FUNCTION_BLOCK TcoDrivesBeckhoffContext EXTENDS TcoCore._internals_TcoContext
VAR
	_callMyPlcInstance 		:	BOOL := FALSE;
	_axis					:	TcoDriveSimpleTest(THIS^);
	_enable					:	BOOL;			
	_enablePositive			:	BOOL;				
	_enableNegative			:	BOOL;        	
	_calibrationCam 		:	BOOL;        	
END_VAR

IF THIS^._callMyPlcInstance THEN
	THIS^.Run();
END_IF

{attribute 'TcRpcEnable'}
METHOD Axis
VAR_INPUT
END_VAR
_axis(	inEnable			:=	_enable, 
		inEnablePositive	:=	_enablePositive, 
		inEnableNegative	:=	_enableNegative, 
		inCalibrationCam	:=	_calibrationCam, 
		inoAxisRef			:=	GVL.Axis1);
END_METHOD

{attribute 'TcRpcEnable'}
METHOD INTERNAL ContextClose
SUPER^._Close();
END_METHOD

{attribute 'TcRpcEnable'}
METHOD INTERNAL ContextOpen
SUPER^._Open();
END_METHOD

METHOD PROTECTED Main
VAR_INPUT
END_VAR
Axis();
END_METHOD

END_FUNCTION_BLOCK

(* stored: Version 1.1.0.1, ProductVersion 3.1.4024.6
   POU TcoDrivesBeckhoffContext: Id {eb079fb3-48a6-04a2-0434-bd84aa928492}, SpecialFunc None
   Method Axis: Id {f8678acb-707d-01d8-2580-87fb1d7a6011}
   Method ContextClose: Id {3c728987-0629-0c84-2598-bb76797d3d61}
   Method ContextOpen: Id {e82e151a-71c2-0de0-0d6a-5bc71438a7cf}
   Method Main: Id {9ed09f46-116f-0806-0bb5-aa63e2f011c3} *)
